PROGRAM PRG_MR5K4_KBO
VAR
    // MR5K4 Flow Press Sensors
    {attribute 'TcLinkTo' := '.fbFlow_1.iRaw := TIIB[EL3054_FWM_PRSM_MR45K4]^AI Standard Channel 3^Value;
                              .fbPress_1.iRaw := TIIB[EL3054_FWM_PRSM_MR45K4]^AI Standard Channel 2^Value
    '}
    {attribute 'pytmc' := '
        pv: MR5K4:KBO
    '}
    fbCoolingPanel : FB_Axilon_Cooling_1f1p;
END_VAR

fbCoolingPanel();

END_PROGRAM

(* stored: Version 1.1.0.1
   POU PRG_MR5K4_KBO: Id {86836c9f-732d-4165-9c34-30c0874932bb}, SpecialFunc None *)
